PROGRAM main
VAR
	MODBEE_HW_INPUTS0 : MODBEE_HW_INPUTS;
	MODBEE_HW_OUTPUTS0 : MODBEE_HW_OUTPUTS;
	start : bool;
	stop : bool;
	run : bool;
	MB_SLAVE_DO : ARRAY [0..31] OF BOOL;
	MB_SLAVE_DI : ARRAY [0..31] OF BOOL;
	MB_WRITE_COILS_DONE : bool;
	MB_READ_COILS_DONE : bool;
	TON0 : TON;
	TON1 : TON;
	TON1_DONE : bool;
	TON0_DONE : bool;
	MB_READ_REGS_DONE : bool;
	MB_SLAVE_AI : ARRAY [0..31] OF INT;
	MB_WRITE_REGS_DONE : bool;
	MB_SLAVE_AO : ARRAY [0..31] OF REAL;
	MB_SLAVE_AO_TEMP : ARRAY [0..31] OF INT;
	MB_WRITE_REGS_DONE0 : bool;
	MODBUS_READ_ARRAY0 : MODBUS_READ_ARRAY;
	MODBUS_READ_ARRAY1 : MODBUS_READ_ARRAY;
	MODBUS_WRITE_ARRAY0 : MODBUS_WRITE_ARRAY;
	MODBUS_WRITE_ARRAY1 : MODBUS_WRITE_ARRAY;
END_VAR

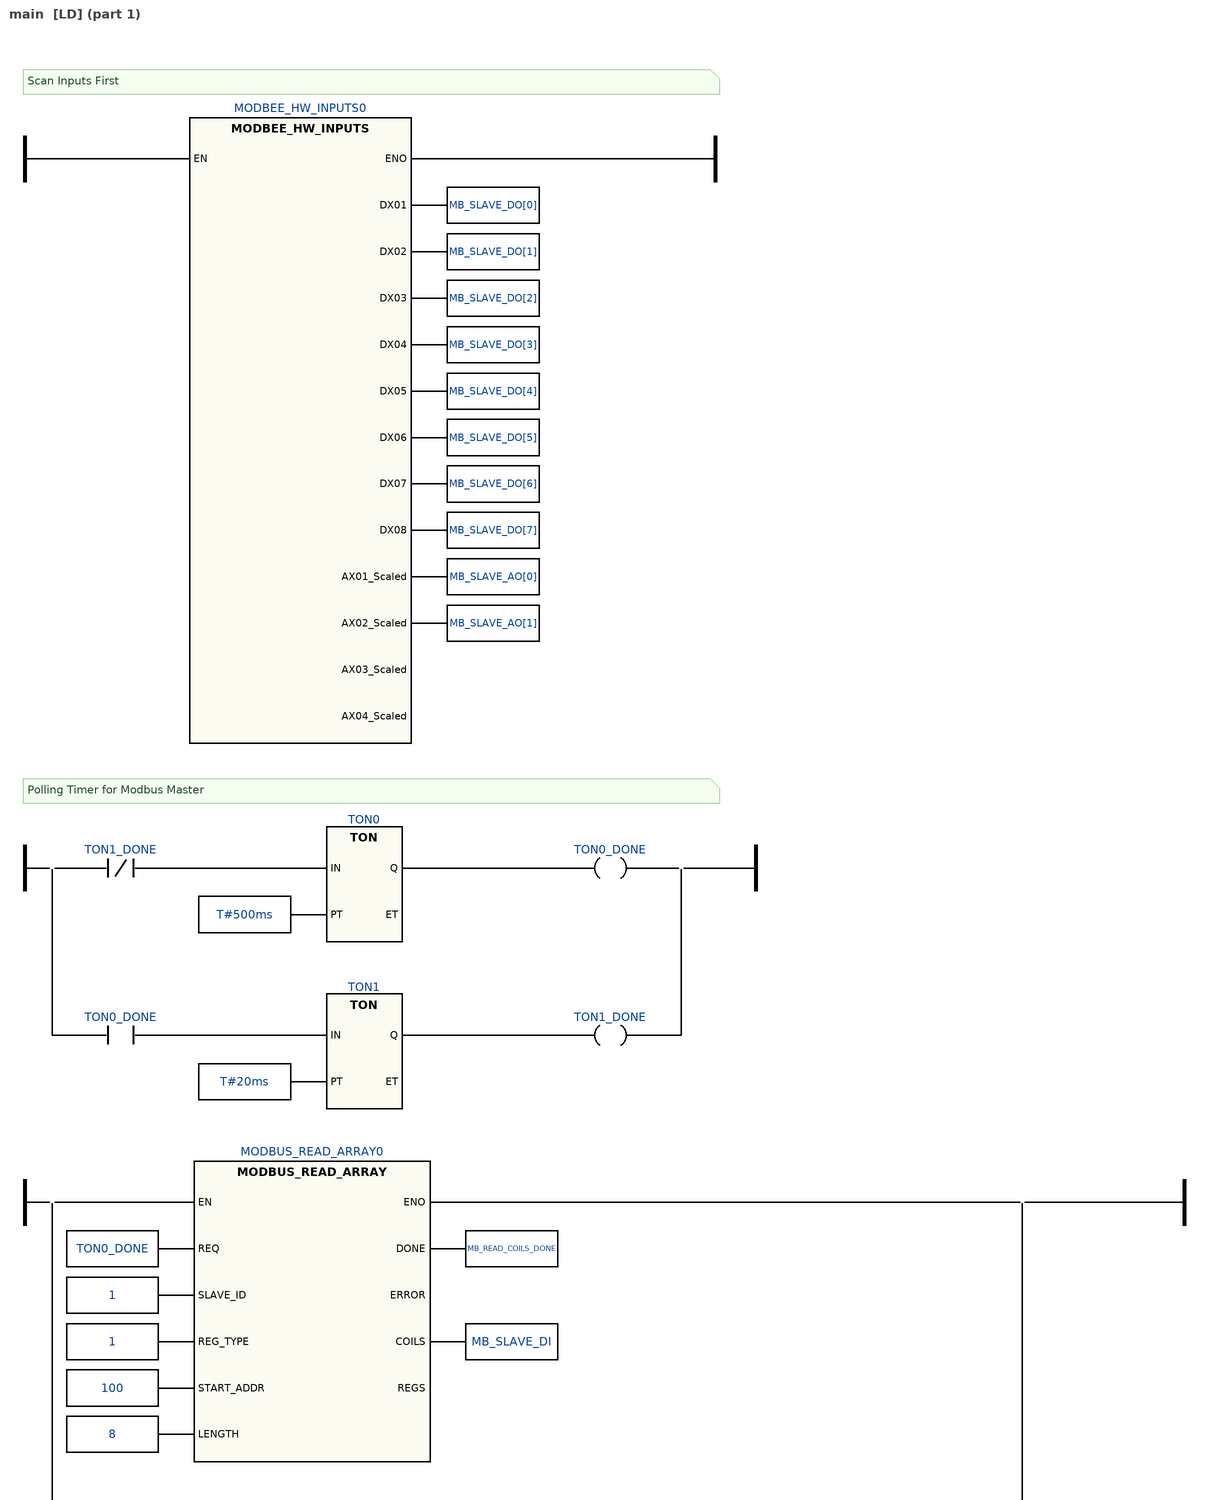
(* LD diagram, written out as Structured Text *)
(* Scan Inputs First *)
MODBEE_HW_INPUTS0();
MB_SLAVE_DO[0] := MODBEE_HW_INPUTS0.DX01;
MB_SLAVE_DO[1] := MODBEE_HW_INPUTS0.DX02;
MB_SLAVE_DO[2] := MODBEE_HW_INPUTS0.DX03;
MB_SLAVE_DO[3] := MODBEE_HW_INPUTS0.DX04;
MB_SLAVE_DO[4] := MODBEE_HW_INPUTS0.DX05;
MB_SLAVE_DO[5] := MODBEE_HW_INPUTS0.DX06;
MB_SLAVE_DO[6] := MODBEE_HW_INPUTS0.DX07;
MB_SLAVE_DO[7] := MODBEE_HW_INPUTS0.DX08;
MB_SLAVE_AO[0] := MODBEE_HW_INPUTS0.AX01_Scaled;
MB_SLAVE_AO[1] := MODBEE_HW_INPUTS0.AX02_Scaled;
(* Polling Timer for Modbus Master *)
TON0(IN := NOT TON1_DONE, PT := T#500ms);
TON0_DONE := TON0.Q;
TON1(IN := TON0_DONE, PT := T#20ms);
TON1_DONE := TON1.Q;
MODBUS_READ_ARRAY0(REQ := TON0_DONE, SLAVE_ID := 1, REG_TYPE := 1, START_ADDR := 100, LENGTH := 8);
MB_READ_COILS_DONE := MODBUS_READ_ARRAY0.DONE;
MB_SLAVE_DI := MODBUS_READ_ARRAY0.COILS;
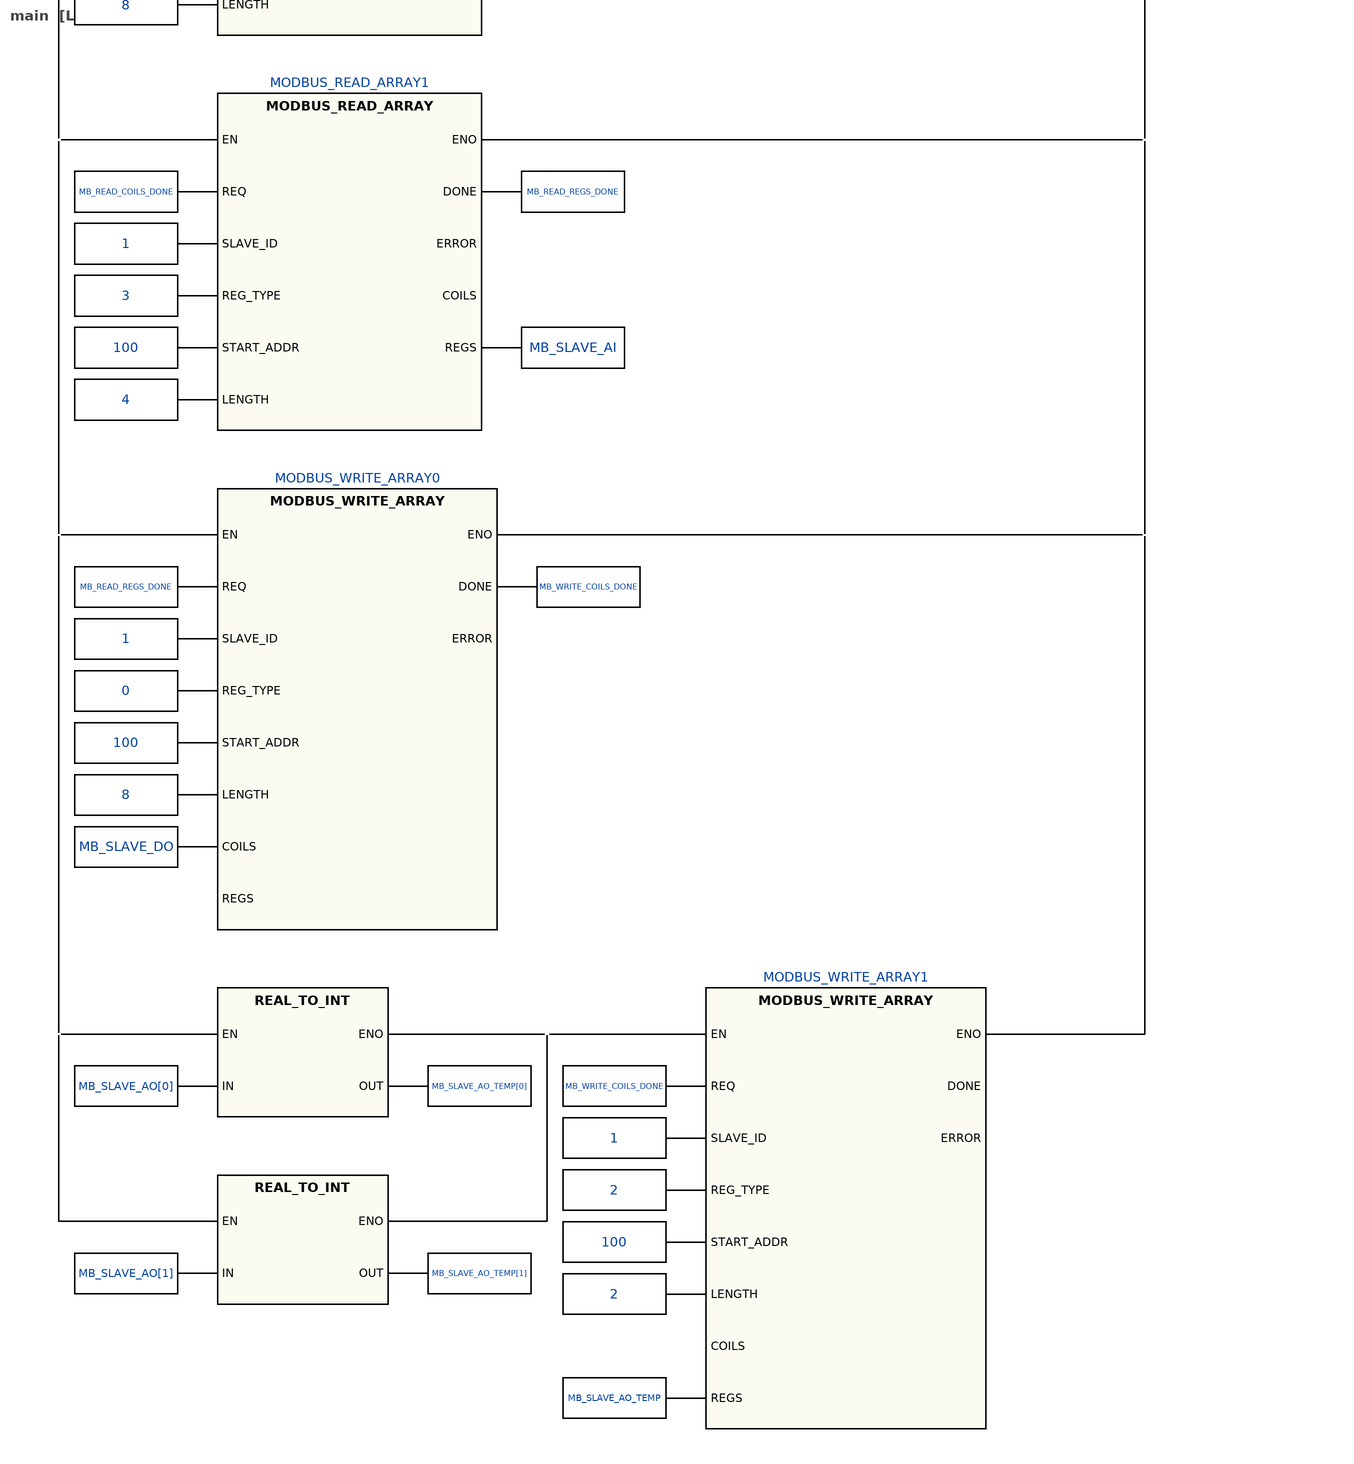
MODBUS_READ_ARRAY1(REQ := MB_READ_COILS_DONE, SLAVE_ID := 1, REG_TYPE := 3, START_ADDR := 100, LENGTH := 4);
MB_READ_REGS_DONE := MODBUS_READ_ARRAY1.DONE;
MB_SLAVE_AI := MODBUS_READ_ARRAY1.REGS;
MODBUS_WRITE_ARRAY0(REQ := MB_READ_REGS_DONE, SLAVE_ID := 1, REG_TYPE := 0, START_ADDR := 100, LENGTH := 8, COILS := MB_SLAVE_DO);
MB_WRITE_COILS_DONE := MODBUS_WRITE_ARRAY0.DONE;
MB_SLAVE_AO_TEMP[0] := REAL_TO_INT(MB_SLAVE_AO[0]);
MB_SLAVE_AO_TEMP[1] := REAL_TO_INT(MB_SLAVE_AO[1]);
MODBUS_WRITE_ARRAY1(REQ := MB_WRITE_COILS_DONE, SLAVE_ID := 1, REG_TYPE := 2, START_ADDR := 100, LENGTH := 2, REGS := MB_SLAVE_AO_TEMP);
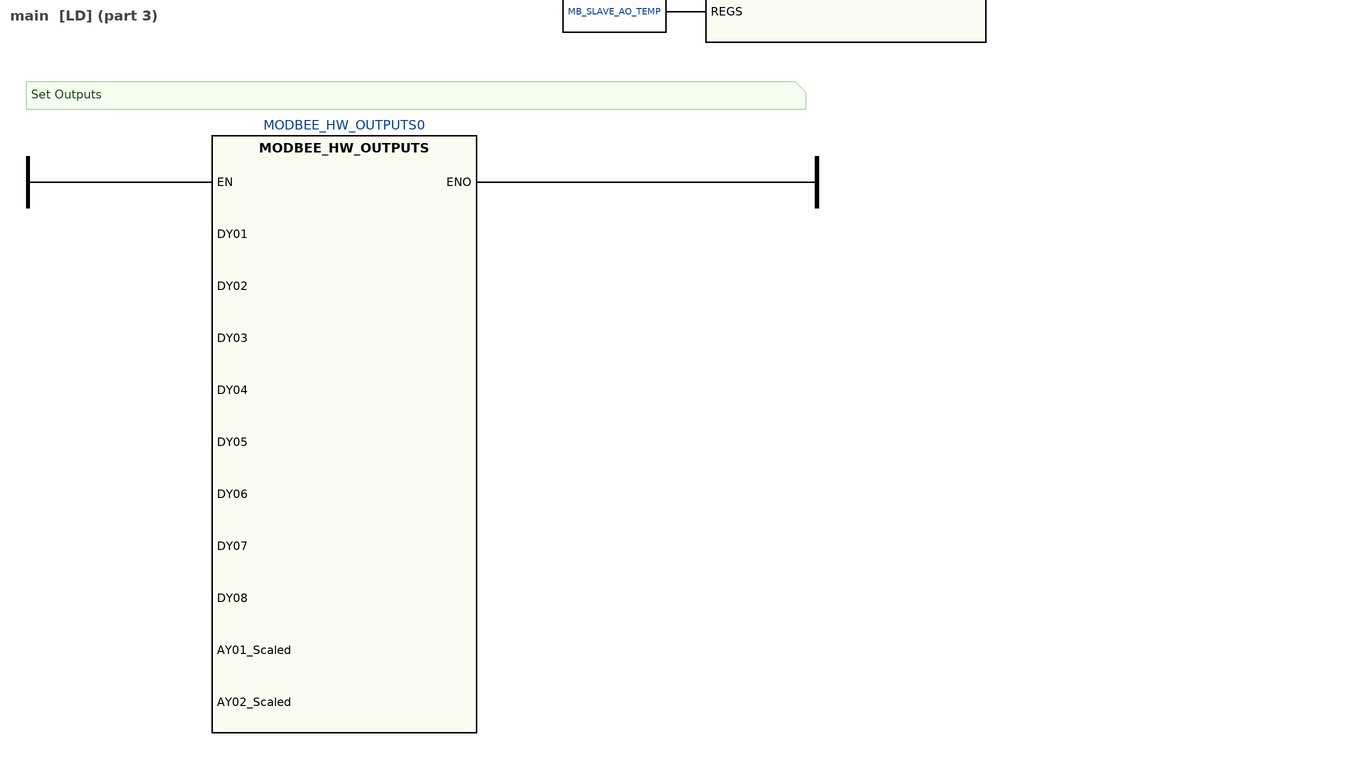
(* Set Outputs *)
MODBEE_HW_OUTPUTS0();
END_PROGRAM
